INTERFACE I_AltAzTelescope EXTENDS I_Telescope

PROPERTY AltitudeOffset : LREAL
GET
END_GET
SET
END_SET
END_PROPERTY

PROPERTY AzimuthOffset : LREAL
GET
END_GET
SET
END_SET
END_PROPERTY

PROPERTY DerotatorOffset : LREAL
GET
END_GET
SET
END_SET
END_PROPERTY

PROPERTY Dut1 : LREAL
GET
END_GET
SET
END_SET
END_PROPERTY

END_INTERFACE

(* stored: Version 1.1.0.1, ProductVersion 3.1.4024.15
   Itf I_AltAzTelescope: Id {eb5dcaf9-36d8-4298-ac4b-d385d1163408}
   Property AltitudeOffset: Id {6e91580b-f921-4d18-9c5d-04331b1b85ef}
   Get Get: Id {91ac621a-2b79-4f9c-89d4-00671a3f53a9}
   Set Set: Id {157ebe42-ab67-47ba-a5c3-03ee2366bfd8}
   Property AzimuthOffset: Id {debc5027-17e9-4739-9a0f-661894e12398}
   Get Get: Id {cfb5cb60-3f07-4c03-ab12-8231c1b5136f}
   Set Set: Id {f8768d35-0d41-490f-9a32-fbbd9836ff1d}
   Property DerotatorOffset: Id {d83deac1-6258-49da-80dc-57a9a51a2246}
   Get Get: Id {639ab416-a7ff-427f-b645-436c0329fb32}
   Set Set: Id {f8869cd1-0209-4ae3-9d27-bb92edf312e5}
   Property Dut1: Id {a3f1c2d4-5e6b-47a8-9c1d-2b3e4f5a6b7c}
   Get Get: Id {b4a2d3e5-6f7c-48b9-ad2e-3c4f5a6b7c8d}
   Set Set: Id {c5b3e4f6-708d-49ca-be3f-4d5a6b7c8d9e} *)
